{attribute 'qualified_only'}
VAR_GLOBAL
	
	// Data to Allen Bradley over EtherNet/IP
	DataEthNetIP_OUTPUT_DINT0				AT%Q*: DINT;
	DataEthNetIP_OUTPUT_DINT1				AT%Q*: DINT;
END_VAR

(* stored: Version 1.1.0.1, ProductVersion 3.1.4024.9
   GVL GVL_outputs: Id {fb385b2f-e42e-4666-9002-a600bc227bd1} *)
